{attribute 'GeneratedUsingTerminal: EK1100-0000-0018'}
{attribute addProperty BoxType "EK1100-0000-0018"}
{attribute addProperty Id "Beckhoff_EJ1xxxEK1122Beckhoff_EJ1xxxEK1122_ACB43C2E15A_0004_EJ1008_0000_0017EJ1008_4201D0AB12A_0005_EJ1128_0000_0016EJ1128_4201D0AB12A_0006_EJ1809_0000_0017EJ1809_FD7895E220A_0007_EJ1819_0000_0017EJ1819_FD7895E220A_0008_EJ1859_0000_0017EJ1859_B9F455E920A_0009_EJ1889_0000_0017EJ1889_FD7895E220A_0003_EJ1122_0000_0016EJ1122_AB5A94672"}
{attribute addProperty CRC "864007402"}
{attribute addProperty Size "121"}
TYPE Beckhoff_EJ1xxx_337FB4EA EXTENDS EK1100_AB5A9467 :
STRUCT
	{attribute addProperty Name "Beckhoff_EJ1xxxEK1122"}
	Beckhoff_EJ1xxxEK1122 : Beckhoff_EJ1xxxEK1122_ACB43C2E;
	{attribute addProperty Name "A_0004_EJ1008_0000_0017"}
	A_0004_EJ1008_0000_0017 : EJ1008_4201D0AB;
	{attribute addProperty Name "A_0005_EJ1128_0000_0016"}
	A_0005_EJ1128_0000_0016 : EJ1128_4201D0AB;
	{attribute addProperty Name "A_0006_EJ1809_0000_0017"}
	A_0006_EJ1809_0000_0017 : EJ1809_FD7895E2;
	{attribute addProperty Name "A_0007_EJ1819_0000_0017"}
	A_0007_EJ1819_0000_0017 : EJ1819_FD7895E2;
	{attribute addProperty Name "A_0008_EJ1859_0000_0017"}
	A_0008_EJ1859_0000_0017 : EJ1859_B9F455E9;
	{attribute addProperty Name "A_0009_EJ1889_0000_0017"}
	A_0009_EJ1889_0000_0017 : EJ1889_FD7895E2;
	{attribute addProperty Name "A_0003_EJ1122_0000_0016"}
	A_0003_EJ1122_0000_0016 : EJ1122_AB5A9467;
END_STRUCT
END_TYPE

(* stored: Version 1.2.0.0, ProductVersion 3.1.4024.9
   DUT Beckhoff_EJ1xxx_337FB4EA: Id {3f58ea71-433c-447c-af71-b7f69bf6e35b} *)
